FUNCTION_BLOCK WORD2WORD (* Simple FB with one algorithm *)
  (* Standard: 61499-1 *)
  (* Version 1.0, 2023-03-07, AK115394 *)
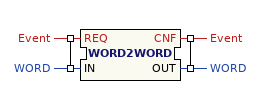
  EVENT_INPUT
    REQ WITH IN; (* Normal Execution Request *)
  END_EVENT
  EVENT_OUTPUT
    CNF WITH OUT; (* Execution Confirmation *)
  END_EVENT
  VAR_INPUT
    IN : WORD;
  END_VAR
  VAR_OUTPUT
    OUT : WORD;
  END_VAR
  ALGORITHM REQ IN ST:
	OUT:=IN;
  END_ALGORITHM
END_FUNCTION_BLOCK
